SUBAPPLICATION RegisterServiceFullOpcUa (* Register a Service using  OPC UA. All possible parameters are available to be set *)
  (* Standard: 61499-2; Description: Copyright (c) 2019 fortiss GmbH This program and the accompanying materials are made available under the terms of the Eclipse Public License 2.0 which is available at https://www.eclipse.org/legal/epl-2.0/ SPDX-License-Identifier: EPL-2.0 *)
  (* Version 1.0, 2019-09-17, Jose Cabral, fortiss GmbH *)
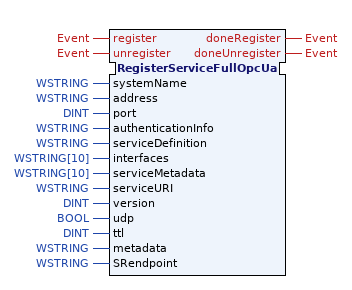
  EVENT_INPUT
    register; (* Register the service *)
    unregister; (* Unregister the service *)
  END_EVENT
  EVENT_OUTPUT
    doneRegister; (* Register finished *)
    doneUnregister; (* Unregister finished *)
  END_EVENT
  VAR_INPUT
    systemName : WSTRING; (* Identification of the system *)
    address : WSTRING; (* Address of the offered services *)
    port : DINT; (* Port of the of the offered services *)
    authenticationInfo : WSTRING; (* Authentication info of the system *)
    serviceDefinition : WSTRING; (* Identification of the service *)
    interfaces : ARRAY [0..9] OF WSTRING; (* Interfaces implemented by the service *)
    serviceMetadata : ARRAY [0..9] OF WSTRING; (* Metadata of the service in key=value format *)
    serviceURI : WSTRING; (* The URL subpath of the Service within the address:port of the Provider *)
    version : DINT; (* The version numbering of the Service provided *)
    udp : BOOL; (* True, if the service is provided via UDP. By default, it is false *)
    ttl : DINT; (* Service validity time period expressed in seconds. This gets converted to a date-time, and stored in the database *)
    metadata : WSTRING; (* Metadata belonging to a service/provider pair *)
    SRendpoint : WSTRING; (* Endpoint (IP:PORT/URI) of the Service Registry *)
  END_VAR
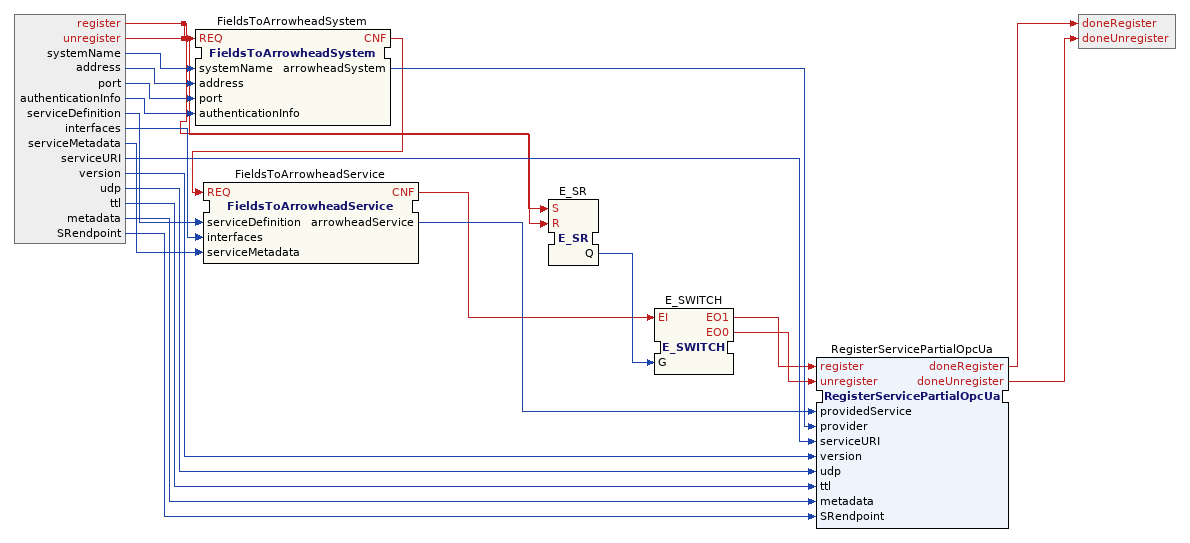
  FBS
    FieldsToArrowheadSystem : FieldsToArrowheadSystem;
    FieldsToArrowheadService : FieldsToArrowheadService;
    E_SR : E_SR;
    E_SWITCH : E_SWITCH;
  END_FBS
  SUBAPPS
    RegisterServicePartialOpcUa : RegisterServicePartialOpcUa;
  END_SUBAPPS
  EVENT_CONNECTIONS
    unregister TO FieldsToArrowheadSystem.REQ;
    register TO FieldsToArrowheadSystem.REQ;
    FieldsToArrowheadSystem.CNF TO FieldsToArrowheadService.REQ;
    register TO E_SR.S;
    unregister TO E_SR.R;
    FieldsToArrowheadService.CNF TO E_SWITCH.EI;
    E_SWITCH.EO1 TO RegisterServicePartialOpcUa.register;
    E_SWITCH.EO0 TO RegisterServicePartialOpcUa.unregister;
    RegisterServicePartialOpcUa.doneRegister TO doneRegister;
    RegisterServicePartialOpcUa.doneUnregister TO doneUnregister;
  END_CONNECTIONS
  DATA_CONNECTIONS
    systemName TO FieldsToArrowheadSystem.systemName;
    address TO FieldsToArrowheadSystem.address;
    port TO FieldsToArrowheadSystem.port;
    authenticationInfo TO FieldsToArrowheadSystem.authenticationInfo;
    serviceDefinition TO FieldsToArrowheadService.serviceDefinition;
    interfaces TO FieldsToArrowheadService.interfaces;
    serviceMetadata TO FieldsToArrowheadService.serviceMetadata;
    E_SR.Q TO E_SWITCH.G;
    FieldsToArrowheadService.arrowheadService TO RegisterServicePartialOpcUa.providedService;
    FieldsToArrowheadSystem.arrowheadSystem TO RegisterServicePartialOpcUa.provider;
    serviceURI TO RegisterServicePartialOpcUa.serviceURI;
    version TO RegisterServicePartialOpcUa.version;
    udp TO RegisterServicePartialOpcUa.udp;
    ttl TO RegisterServicePartialOpcUa.ttl;
    metadata TO RegisterServicePartialOpcUa.metadata;
    SRendpoint TO RegisterServicePartialOpcUa.SRendpoint;
  END_CONNECTIONS
END_SUBAPPLICATION
